// TIA Portal V20 export
DATA_BLOCK "CallEquipment_DB"   // DB196
{ DB_Accessible_From_OPC_UA := 'FALSE' }
// stored: AssignedProDiagFB Unit1.Em3.ProDiag, DBAccessibleFromOPCUA false, DBAccessibleFromWebserver false, InstanceOfName Unit1.Em3.CallEquipment, InstanceOfType FB, Namespace Unit1.Em3
"Unit1.Em3.CallEquipment"
   // VAR_INPUT
   //    ZoneOperationEnable { ExternalWritable := 'False'} : "LWONIK_typeSafetyZoneManualOperation";
   //    unitEnableControlInterfaces { ExternalWritable := 'False'} : "LAF_typeEnableControlInterfaces";
   //    commandExcute { ExternalWritable := 'False'} : Bool;
   // END_VAR
   // VAR_IN_OUT
   //    unitStatus : "LAF_typeUnitStatus";
   //    emFeedback : "LUC_typeEmFeedback";
   //    unitAlarmDB : "LAF_typeAlarms";
   // END_VAR
   // VAR
   //    instSequenceWebGuid { ExternalWritable := 'False'} : "Unit1.Em3.Sequence_1_WebGuid";
   //    instWebGuidInitializedJob1 { ExternalWritable := 'False'} : "LAF_SelectJob";
   //    instWebGuidMotionCalculateJob2 { ExternalWritable := 'False'} : "LAF_SelectJob";
   //    instWebGuidMotionOneCellJob3 { ExternalWritable := 'False'} : "LAF_SelectJob";
   //    instWebGuidMotionFullStepJob4 { ExternalWritable := 'False'} : "LAF_SelectJob";
   //    instWebGuidMotionAutoJob5 { ExternalWritable := 'False'} : "LAF_SelectJob";
   //    instWebGuidMotionSemiStepJob6 { ExternalWritable := 'False'} : "LAF_SelectJob";
   //    instWebGuidMotionCycleStopJob7 { ExternalWritable := 'False'} : "LAF_SelectJob";
   //    instWebGuidMotionFastStopJob8 { ExternalWritable := 'False'} : "LAF_SelectJob";
   //    instCmMasterVirtualAxis { ExternalWritable := 'False'} : "LBC_AxisControl_TecPlcCn";
   //    instCmUnwinderVirtualAxis { ExternalWritable := 'False'} : "LBC_AxisControl_TecPlcCn";
   //    instCmDancerRegulatorOnOff { ExternalWritable := 'False'} : "LBC_TwoWayActuatorCn";
   //    instCmDancerSafetyPinIdlePosition { ExternalWritable := 'False'} : "LBC_DigitalSignalCn";
   //    instCmDancerEncoderAnalogInput { ExternalWritable := 'False'} : "LBC_AnalogInputCn";
   //    instCmLoadCellAnalogInput { ExternalWritable := 'False'} : "LBC_AnalogInputCn";
   //    instCmDancerElectroPneumaticRegulatorAnalogOutput { ExternalWritable := 'False'} : "LBC_AnalogOutputCn";
   //    instCmWebGuideEpc { ExternalWritable := 'False'} : "LER_EPC_CON600";
   //    instCmMasterAxisControlInterlockSummary { ExternalWritable := 'False'} : "LER_AxisControl_InterlockSummary";
   //    instCmUnwinderAxisControlInterlockSummary { ExternalWritable := 'False'} : "LER_AxisControl_InterlockSummary";
   //    statUnitStatus { ExternalWritable := 'False'} : "LAF_typeUnitStatus";
   //    instManageAlarms { ExternalWritable := 'False'} : "LAF_ManageAlarms";
   //    instEventsPFE { S7_SetPoint := 'True'} : "Unit1.Em3.EventsPFE";
   //    statLoadcellBuf { ExternalWritable := 'False'} : Int;
   //    statEnableManualCmds { ExternalWritable := 'False'} : Bool;
   //    statPulse { ExternalWritable := 'False'} : Array[0..99] of Bool;
   //    statTonTimer { ExternalWritable := 'False'} : Array[0..99] of TON_TIME;
   //    statTofTimer { ExternalWritable := 'False'} : Array[0..99] of TOF_TIME;
   //    instCheckCamRecipeChanged { ExternalWritable := 'False'} : "LER_CheckCamRecipeChanged";
   //    statCheckCamRecipeChangedStatus { ExternalWritable := 'False'} : Struct
   //       ValidParameters : Bool;
   //       ParameterChanged : Bool;
   //       ExecuteRequired : Bool;
   //    END_STRUCT;
   //    NGConveyorFull { ExternalVisible := 'False'; ExternalWritable := 'False'} : Bool;
   //    Stack1ConveyorFull { ExternalVisible := 'False'; ExternalWritable := 'False'} : Bool;
   //    Stack2ConveyorFull { ExternalVisible := 'False'; ExternalWritable := 'False'} : Bool;
   //    All_Full { ExternalVisible := 'False'; ExternalWritable := 'False'} : Bool;
   //    Stack1_Full_Abnormal { ExternalVisible := 'False'; ExternalWritable := 'False'} : Bool;
   //    Stack2_Full_Abnormal { ExternalVisible := 'False'; ExternalWritable := 'False'} : Bool;
   //    CutConveyorFull { ExternalVisible := 'False'; ExternalWritable := 'False'} : Bool;
   //    "Stack#1BA030Unuse" { ExternalVisible := 'False'; ExternalWritable := 'False'} : Bool;
   //    "Stack#2BA040Unuse" { ExternalVisible := 'False'; ExternalWritable := 'False'} : Bool;
   //    instCVFullChargeCheckCMD { S7_SetPoint := 'True'} : "LAF_SelectJob";
   //    CellCountDiv1 { S7_SetPoint := 'True'} : LReal;
   //    CellCountDiv2 { S7_SetPoint := 'True'} : LReal;
   // END_VAR
BEGIN
END_DATA_BLOCK
